Staubli VAL3: getStrSign.pgx

program getStrSign(string x_sText (dimensions=1), string& x_sStrSign[] (dimensions=1))
begin
  //分割"="前后的字符串，保存至x_sStrSign字符串数组中
  //获取"="前面的标识字符串
  call split(x_sText,"=",x_sStrSign)
end
